// TIA Portal V19 export
TYPE "PathTestHMI"
// stored: Access Published
   STRUCT
      ManCmdStartTest : Bool;
      TestEnabled : Bool;
      TestRequired : Bool;
      TestStarted : Bool;
      TestRunning : Bool;
   END_STRUCT;
END_TYPE
